Fanuc KAREL source: kt00070.KL

-- PROVISIONAL review KL for V1013-1; original PC SHA256 691aab5e7a6ece47d869c460b327f1d9b14c305389742d016a4ad6dd2edd2b84
-- Incomplete behavior may be omitted. Consult companion uncertainty JSON. Do not deploy.
PROGRAM KT00070
%NOLOCKGROUP
VAR
  I1 : INTEGER
  OUT : REAL
-- UNRESOLVED_DECL Y2 type=002018
BEGIN
  -- UNRESOLVED_PC offsets 5-16; opcodes 2E,23
  -- UNRESOLVED_PC offsets 21-35; opcodes 2E,22,9D,33,B2
  -- UNRESOLVED_PC offsets 40-63; opcodes 21,22,9D,33,B1,54,64,23
  -- UNRESOLVED_PC offsets 68-72; opcodes 7F
END KT00070
